// TIA Portal V20 export
DATA_BLOCK "EmNodes"   // DB3
{ DB_Accessible_From_OPC_UA := 'FALSE' }
AUTHOR : ERsystem_FA2_DH. Kim
// stored: Access Published, DBAccessibleFromOPCUA false, DBAccessibleFromWebserver false, MemoryReserve 100, Namespace Unit1
   VAR
      unitStatus { ExternalWritable := 'False'} : "LAF_typeUnitStatus";   // Status of the unit
      emFeedback { ExternalWritable := 'False'} : Array[0.._.U1_NO_OF_EMs] of "LUC_typeEmFeedback";   // Status of the individual equipment modules
      emRelations : Struct
         em00 : "Unit1.type_emRelations_em0";
         em01 : "Unit1.type_emRelations_em1";
         em02 : "Unit1.type_emRelations_em2";
         em03 : "Unit1.type_emRelations_em3";
         em04 : "Unit1.type_emRelations_em4";
         em05 : "Unit1.type_emRelations_em5";
         em06 : "Unit1.type_emRelations_em6";
         em07 : "Unit1.type_emRelations_em7";
      END_STRUCT;
      emIt { S7_SetPoint := 'True'} : Array[0..13] of "LER_OEM_Data";
      enableControlInterfaces { ExternalWritable := 'False'} : "LAF_typeEnableControlInterfaces";
      oem { ExternalAccessible := 'False'; ExternalVisible := 'False'; ExternalWritable := 'False'; S7_SetPoint := 'True'} : Array[0..10] of "LER_OEM_Data";
      FATModeSelect { ExternalWritable := 'False'} : "LER_TypeFATMode_ModeSelect";
   END_VAR
   VAR RETAIN
      FATModeInterface { ExternalWritable := 'False'} : "LER_TypeFATModeInterface";
   END_VAR
   VAR
      signalStack { ExternalWritable := 'False'} : "LUC_typeSignalStackByBool";
      clock { ExternalWritable := 'False'} : "LAF_typeGlobalClockMem";
      slmRunning { S7_SetPoint := 'True'} : Bool;
      slmPowerOff { ExternalWritable := 'False'} : Bool;
      InterfaceTestMode { ExternalWritable := 'False'} : Bool;
      CapabilityModeComplete { ExternalWritable := 'False'} : Bool;
      SamplingModeComplete { ExternalWritable := 'False'} : Bool;
      stateCommandsExecute { ExternalWritable := 'False'} : Bool;
      atLeastOneDoorUnlock { ExternalWritable := 'False'} : Bool;
      SleepModeActivationTime : Time;
      DeepSleepModeActivationTime : Time;
      SleepModeChangeReq : Bool;
      DeepSleepModeChangeReq : Bool;
      WakeupRecoveryRequired : Bool;
      sleep : Struct
         State { S7_SetPoint := 'True'} : "LER_typeSleepMode";
         command { S7_SetPoint := 'True'} : "LER_typeSleep";
      END_STRUCT;
      "========Communication========" { ExternalWritable := 'False'} : Bool;
      BA010 { ExternalWritable := 'False'} : "LER_typeCommunicationReelCut";
      BA015 { ExternalWritable := 'False'} : "LER_typeCommunicationReelCut";
      BA040 { ExternalWritable := 'False'} : "LER_typeCommunicationStack";
      BA060 { S7_SetPoint := 'True'} : "LER_typeCommunicationInspection";
      "========Safety========" { ExternalWritable := 'False'} : Bool;
      devicesSummary : "LWONIK_typeDevicesStatusSummary";
      safetyZone1OpEnable { ExternalWritable := 'False'} : "LWONIK_typeSafetyZoneManualOperation";
      safetyZone2OpEnable { ExternalWritable := 'False'} : "LWONIK_typeSafetyZoneManualOperation";
      safetyZone3OpEnable { ExternalWritable := 'False'} : "LWONIK_typeSafetyZoneManualOperation";
      doorOpenRequest : Bool;
      safetyStatusZone1 { S7_SetPoint := 'True'} : "LWONIK_typeZoneStatus";
      safetyStatusZone2 { S7_SetPoint := 'True'} : "LWONIK_typeZoneStatus";
      safetyStatusZone3 { S7_SetPoint := 'True'} : "LWONIK_typeZoneStatus";
      mainOpMode : "LWONIK_typeOperationMode";
      pHmiMode { ExternalWritable := 'False'} : "LWONIK_typePhmiMode";
      scsMode { ExternalWritable := 'False'} : "LWONIK_typeScsMode";
      rcMode1 { S7_SetPoint := 'True'} : "LWONIK_typeRollChangeMode";
      rcMode2 { S7_SetPoint := 'True'} : "LWONIK_typeRollChangeMode";
      scrapBox1 { S7_SetPoint := 'True'} : "LWONIK_typeScrapBox";
      scrapBox2 { S7_SetPoint := 'True'} : "LWONIK_typeScrapBox";
      SafetySensor { S7_SetPoint := 'True'} : "LWONIK_typeSafetySensor";
      EstopStatus { ExternalWritable := 'False'} : "LWONIK_typeFromSafetyEstopStatus";
      FdoorStatus { ExternalWritable := 'False'} : "LWONIK_typeFromSafetyDoorStatus";
      fDoorDrive : "Safety.typeFDoorFunction";
      cvCoverStatus : Struct
         cvCoverOK1 { ExternalWritable := 'False'} : Bool;
         cvCoverOK2 { ExternalWritable := 'False'} : Bool;
         cvCoverAllOK { ExternalWritable := 'False'} : Bool;
         cvCoverSystemFaults { ExternalWritable := 'False'} : Bool;
      END_STRUCT;
      AllSFDoorOpen { S7_SetPoint := 'True'} : Bool;
      AllFDoorClosed : Bool;
      OpHmiOperationEnable : Bool;
      PHmiOperationEnable : Bool;
      MobilePanelConnected : Bool;
      MobilePanelPermissions : Bool;
      BA60ExternalDoorOpen : Bool;
      SS1TimeExtension : Bool;
      EnableServoAck : Bool;
      BA10SCSModeSelect : Bool;
      BA15SCSModeSelect : Bool;
      BA40SCSModeSelect : Bool;
      BA60SCSModeSelect : Bool;
      BA60LightCurtainMutingOn : Bool;
      "=======ETC========" : Bool;
      allBrakeTest { ExternalWritable := 'False'} : "LER_typeBrakeTestUnitInterface";
      booltest { S7_SetPoint := 'True'} : Array[0..15] of Bool;
      motionInterface : Struct
         Dancer : Struct
            Enable : Bool := FALSE;
            Stop : Bool := FALSE;
            Reset : Bool := FALSE;
         END_STRUCT;
         StackMain : Struct
            Calculate { ExternalAccessible := 'False'; ExternalVisible := 'False'; ExternalWritable := 'False'} : Bool;
            SemiStep { ExternalAccessible := 'False'; ExternalVisible := 'False'; ExternalWritable := 'False'} : Bool;
            FullStep { ExternalAccessible := 'False'; ExternalVisible := 'False'; ExternalWritable := 'False'} : Bool;
            SepaClean { ExternalAccessible := 'False'; ExternalVisible := 'False'; ExternalWritable := 'False'} : Bool;
            Auto { ExternalAccessible := 'False'; ExternalVisible := 'False'; ExternalWritable := 'False'} : Bool;
            StopMotion { ExternalAccessible := 'False'; ExternalVisible := 'False'; ExternalWritable := 'False'} : Bool;
            Reset { ExternalAccessible := 'False'; ExternalVisible := 'False'; ExternalWritable := 'False'} : Bool;
         END_STRUCT;
      END_STRUCT;
      FullStepRun : Bool;
      MotionRunlockBit : Bool;
      FullStepReady : Bool;
      MotionReady : Bool;
      SpecialFunctionEnable : Bool;
   END_VAR
BEGIN
   // emRelations.em04."Bool"[10] : EM4 Motion Ready / No Job Active
   // emRelations.em04.sequence.Spare1.preOperationCheck.Bool12 : EM4 Ready For Motion
   // emRelations.em05."Bool"[10] : EM5 Motion Ready / No Job Active
   // emRelations.em05.sequence.Spare1.preOperationCheck.Bool12 : EM5 Ready For Motion
   // emRelations.em06.sequence.Spare1.preOperationCheck.Bool12 : EM6 Ready For Motion
   // emRelations.em06.sequence.Spare1.jobInterface[14].motionRequest : SepaCleanMotion Request
   // emRelations.em07."Bool"[1] : SepaGirpperAxisX Move To BA60
   // BA010.ReelCutToStack.InterfaceData."Bool"[0] : Load Enable
   // BA010.ReelCutToStack.InterfaceData."Bool"[1] : Load Complete Comfirm
   // BA010.ReelCutToStack.InterfaceData."Bool"[2] : Cell Data Report
   // BA010.ReelCutToStack.InterfaceData."Bool"[10] : CollisionAreaOn
   // BA010.ReelCutToStack.InterfaceData."Bool"[11] : CollisionAreaOff
   // BA010.ReelCutToStack.InterfaceData."Bool"[20] : Motion Ready
   // BA010.ReelCutToStack.InterfaceData."Bool"[21] : Motion Auto Standby
   // BA010.ReelCutToStack.InterfaceData."Bool"[22] : Motion Auto Mode
   // BA010.ReelCutToStack.InterfaceData."Bool"[23] : Motion Stop CMD (Motion Stop Req)
   // BA010.ReelCutToStack.InterfaceData."Bool"[30] : HoursTestMode.On/Off.Status (ReelCut)
   // BA010.ReelCutToStack.InterfaceData."Bool"[31] : HourTestMode_Completed (ReelCut)
   // BA010.ReelCutToStack.InterfaceData."Bool"[32] : CapabilityMode.On/Off.Status (ReelCut)
   // BA010.ReelCutToStack.InterfaceData."Bool"[33] : CapabilityMode_Completed (ReelCut)
   // BA010.ReelCutToStack.InterfaceData."Bool"[34] : FATMode.Apply (ReelCut)
   // BA010.ReelCutToStack.InterfaceData.LReal[10] : Select Hours (ReelCut)
   // BA010.StackToReelCut.InterfaceData."Bool"[0] : From Load Requset
   // BA010.StackToReelCut.InterfaceData."Bool"[1] : From Load Busy
   // BA010.StackToReelCut.InterfaceData."Bool"[2] : From Load Complete
   // BA010.StackToReelCut.InterfaceData."Bool"[3] : Cell Data Request
   // BA010.StackToReelCut.InterfaceData."Bool"[4] : Cell Data Report Ack
   // BA010.StackToReelCut.InterfaceData."Bool"[5] : Cell Data Report Nck
   // BA010.StackToReelCut.InterfaceData."Bool"[10] : Stack#1 Gauge RnR Complete
   // BA010.StackToReelCut.InterfaceData."Bool"[15] : HeartBeat
   // BA010.StackToReelCut.InterfaceData."Bool"[19] : From Stack#1 Count Mismatch Call
   // BA010.StackToReelCut.InterfaceData."Bool"[20] : From Motion Ready Status (Stack#1 Full)
   // BA010.StackToReelCut.InterfaceData."Bool"[21] : From Stack#1 in Motion Auto Standby
   // BA010.StackToReelCut.InterfaceData."Bool"[22] : From Stack#1 in Motion Auto Mode
   // BA010.StackToReelCut.InterfaceData."Bool"[23] : From Motion Start CMD (Stack#1 Motion Req)
   // BA010.StackToReelCut.InterfaceData."Bool"[24] : From Motion Stop CMD (Stack#1 Error)
   // BA010.StackToReelCut.InterfaceData."Bool"[25] : From Stack#1 Unloading
   // BA010.StackToReelCut.InterfaceData."Bool"[26] : From Stack#1 Loading Ok
   // BA010.StackToReelCut.InterfaceData."Bool"[30] : HoursTestMode.On/Off.Status (STK)
   // BA010.StackToReelCut.InterfaceData."Bool"[31] : HourTestMode_Completed (STK)
   // BA010.StackToReelCut.InterfaceData."Bool"[32] : CapabilityMode.On/Off.Status (STK)
   // BA010.StackToReelCut.InterfaceData."Bool"[33] : CapabilityMode_Completed (STK)
   // BA010.StackToReelCut.InterfaceData."Bool"[34] : FATMode.Apply (STK)
   // BA010.StackToReelCut.InterfaceData."Bool"[40] : HoursTestMode.On/Off.Status (INS)
   // BA010.StackToReelCut.InterfaceData."Bool"[41] : HourTestMode_Completed (INS)
   // BA010.StackToReelCut.InterfaceData."Bool"[42] : CapabilityMode.On/Off.Status (INS)
   // BA010.StackToReelCut.InterfaceData."Bool"[43] : CapabilityMode_Completed (INS)
   // BA010.StackToReelCut.InterfaceData."Bool"[44] : FATMode.Apply (INS)
   // BA010.StackToReelCut.InterfaceData.LReal[0] : From Stack#1 Cell Count
   // BA010.StackToReelCut.InterfaceData.LReal[1] : From Stack#1 CPM
   // BA010.StackToReelCut.InterfaceData.LReal[2] : Stack#1 Gauge RnR3 Mode Count
   // BA010.StackToReelCut.InterfaceData.LReal[10] : Select Hours (STK)
   // BA010.StackToReelCut.InterfaceData.LReal[11] : Select Hours (INS)
   // BA015.ReelCutToStack.InterfaceData."Bool"[0] : Load Enable
   // BA015.ReelCutToStack.InterfaceData."Bool"[1] : Load Complete Comfirm
   // BA015.ReelCutToStack.InterfaceData."Bool"[2] : Cell Data Report
   // BA015.ReelCutToStack.InterfaceData."Bool"[10] : CollisionAreaOn
   // BA015.ReelCutToStack.InterfaceData."Bool"[11] : CollisionAreaOff
   // BA015.ReelCutToStack.InterfaceData."Bool"[20] : Motion Ready
   // BA015.ReelCutToStack.InterfaceData."Bool"[21] : Motion Auto Standby
   // BA015.ReelCutToStack.InterfaceData."Bool"[22] : Motion Auto Mode
   // BA015.ReelCutToStack.InterfaceData."Bool"[23] : Motion Stop CMD (Motion Stop Req)
   // BA015.ReelCutToStack.InterfaceData."Bool"[30] : HoursTestMode.On/Off.Status (ReelCut)
   // BA015.ReelCutToStack.InterfaceData."Bool"[31] : HourTestMode_Completed (ReelCut)
   // BA015.ReelCutToStack.InterfaceData."Bool"[32] : CapabilityMode.On/Off.Status (ReelCut)
   // BA015.ReelCutToStack.InterfaceData."Bool"[33] : CapabilityMode_Completed (ReelCut)
   // BA015.ReelCutToStack.InterfaceData."Bool"[34] : FATMode.Apply (ReelCut)
   // BA015.ReelCutToStack.InterfaceData.LReal[10] : Select Hours (ReelCut)
   // BA015.StackToReelCut.InterfaceData."Bool"[0] : From Load Requset
   // BA015.StackToReelCut.InterfaceData."Bool"[1] : From Load Busy
   // BA015.StackToReelCut.InterfaceData."Bool"[2] : From Load Complete
   // BA015.StackToReelCut.InterfaceData."Bool"[3] : Cell Data Request
   // BA015.StackToReelCut.InterfaceData."Bool"[4] : Cell Data Report Ack
   // BA015.StackToReelCut.InterfaceData."Bool"[5] : Cell Data Report Nck
   // BA015.StackToReelCut.InterfaceData."Bool"[10] : Stack#1 Gauge RnR Complete
   // BA015.StackToReelCut.InterfaceData."Bool"[15] : HeartBeat
   // BA015.StackToReelCut.InterfaceData."Bool"[19] : From Stack#1 Count Mismatch Call
   // BA015.StackToReelCut.InterfaceData."Bool"[20] : From Motion Ready Status (Stack#1 Full)
   // BA015.StackToReelCut.InterfaceData."Bool"[21] : From Stack#1 in Motion Auto Standby
   // BA015.StackToReelCut.InterfaceData."Bool"[22] : From Stack#1 in Motion Auto Mode
   // BA015.StackToReelCut.InterfaceData."Bool"[23] : From Motion Start CMD (Stack#1 Motion Req)
   // BA015.StackToReelCut.InterfaceData."Bool"[24] : From Motion Stop CMD (Stack#1 Error)
   // BA015.StackToReelCut.InterfaceData."Bool"[25] : From Stack#1 Unloading
   // BA015.StackToReelCut.InterfaceData."Bool"[26] : From Stack#1 Loading Ok
   // BA015.StackToReelCut.InterfaceData."Bool"[30] : HoursTestMode.On/Off.Status (STK)
   // BA015.StackToReelCut.InterfaceData."Bool"[31] : HourTestMode_Completed (STK)
   // BA015.StackToReelCut.InterfaceData."Bool"[32] : CapabilityMode.On/Off.Status (STK)
   // BA015.StackToReelCut.InterfaceData."Bool"[33] : CapabilityMode_Completed (STK)
   // BA015.StackToReelCut.InterfaceData."Bool"[34] : FATMode.Apply (STK)
   // BA015.StackToReelCut.InterfaceData."Bool"[40] : HoursTestMode.On/Off.Status (INS)
   // BA015.StackToReelCut.InterfaceData."Bool"[41] : HourTestMode_Completed (INS)
   // BA015.StackToReelCut.InterfaceData."Bool"[42] : CapabilityMode.On/Off.Status (INS)
   // BA015.StackToReelCut.InterfaceData."Bool"[43] : CapabilityMode_Completed (INS)
   // BA015.StackToReelCut.InterfaceData."Bool"[44] : FATMode.Apply (INS)
   // BA015.StackToReelCut.InterfaceData.LReal[0] : From Stack#1 Cell Count
   // BA015.StackToReelCut.InterfaceData.LReal[1] : From Stack#1 CPM
   // BA015.StackToReelCut.InterfaceData.LReal[2] : Stack#1 Gauge RnR3 Mode Count
   // BA015.StackToReelCut.InterfaceData.LReal[10] : Select Hours (STK)
   // BA015.StackToReelCut.InterfaceData.LReal[11] : Select Hours (INS)
   // BA060.InspectionToStack.InterfaceData."Bool"[0] : Heartbeat
   // BA060.InspectionToStack.InterfaceData."Bool"[1] : ReadyForOperation
   // BA060.InspectionToStack.InterfaceData."Bool"[2] : ReachedHome
   // BA060.InspectionToStack.InterfaceData."Bool"[3] : MachineInOperation
   // BA060.InspectionToStack.InterfaceData."Bool"[4] : LoaderOutsideModule
   // BA060.InspectionToStack.InterfaceData."Bool"[5] : LoaderOutsideCollision
   // BA060.InspectionToStack.InterfaceData."Bool"[10] : PartClamped
   // BA060.InspectionToStack.InterfaceData."Bool"[11] : PartUnclamped
   // BA060.InspectionToStack.InterfaceData."Bool"[16] : RequestUnclamp
   // BA060.InspectionToStack.InterfaceData."Bool"[17] : PartOn
   // BA060.InspectionToStack.InterfaceData."Bool"[18] : RequestPart
   // BA060.InspectionToStack.InterfaceData."Bool"[19] : OnPositionUnloading
   // BA060.InspectionToStack.InterfaceData."Bool"[22] : RequestCollisionON
   // BA060.InspectionToStack.InterfaceData."Bool"[23] : UnoadComplete
   // BA060.InspectionToStack.InterfaceData."Bool"[26] : DataCatchUp
   // BA060.InspectionToStack.InterfaceData."Bool"[27] : DataCompareOK
   // BA060.InspectionToStack.InterfaceData."Bool"[28] : DataDeleted
   // BA060.InspectionToStack.InterfaceData."Bool"[32] : NG RequestPart
   // BA060.InspectionToStack.InterfaceData."Bool"[33] : NG RequestUnclamp
   // BA060.InspectionToStack.InterfaceData."Bool"[34] : NG UnoadComplete
   // BA060.InspectionToStack.InterfaceData."Bool"[40] : HoursTestMode.On/Off.Status (INS)
   // BA060.InspectionToStack.InterfaceData."Bool"[41] : HourTestMode_Completed (INS)
   // BA060.InspectionToStack.InterfaceData."Bool"[42] : CapabilityMode.On/Off.Status (INS)
   // BA060.InspectionToStack.InterfaceData."Bool"[43] : CapabilityMode_Completed (INS)
   // BA060.InspectionToStack.InterfaceData."Bool"[44] : FATMode.Apply (INS)
   // BA060.InspectionToStack.InterfaceData."Bool"[48] : ReturnToHome
   // BA060.InspectionToStack.InterfaceData."Bool"[49] : AutoStart
   // BA060.InspectionToStack.InterfaceData."Bool"[50] : EndOfCycle
   // BA060.InspectionToStack.InterfaceData."Bool"[51] : RequestGateOpen
   // BA060.InspectionToStack.InterfaceData.LReal[0] : Select Hours (INS)
   // BA060.StackToInspection.InterfaceData."Bool"[0] : Heartbeat
   // BA060.StackToInspection.InterfaceData."Bool"[1] : ReadyForOperation
   // BA060.StackToInspection.InterfaceData."Bool"[2] : ReachedHome
   // BA060.StackToInspection.InterfaceData."Bool"[3] : MachineInOperation
   // BA060.StackToInspection.InterfaceData."Bool"[4] : NoInterference
   // BA060.StackToInspection.InterfaceData."Bool"[10] : PartClamped
   // BA060.StackToInspection.InterfaceData."Bool"[11] : PartUnclamped
   // BA060.StackToInspection.InterfaceData."Bool"[16] : RequestClamp
   // BA060.StackToInspection.InterfaceData."Bool"[17] : PartOn
   // BA060.StackToInspection.InterfaceData."Bool"[18] : PartReady
   // BA060.StackToInspection.InterfaceData."Bool"[19] : LoaderInTranferArea
   // BA060.StackToInspection.InterfaceData."Bool"[20] : CollisionAreaOn
   // BA060.StackToInspection.InterfaceData."Bool"[21] : CollisionAreaOff
   // BA060.StackToInspection.InterfaceData."Bool"[23] : LoadComplete
   // BA060.StackToInspection.InterfaceData."Bool"[26] : DataCatchUp
   // BA060.StackToInspection.InterfaceData."Bool"[27] : DataCompareOK
   // BA060.StackToInspection.InterfaceData."Bool"[28] : DataDeleted
   // BA060.StackToInspection.InterfaceData."Bool"[32] : NG PartReady
   // BA060.StackToInspection.InterfaceData."Bool"[33] : NG RequestClamp
   // BA060.StackToInspection.InterfaceData."Bool"[34] : NG LoadComplete
   // BA060.StackToInspection.InterfaceData."Bool"[35] : HoursTestMode.On/Off.Status (ReelCut)
   // BA060.StackToInspection.InterfaceData."Bool"[36] : HourTestMode_Completed (ReelCut)
   // BA060.StackToInspection.InterfaceData."Bool"[37] : CapabilityMode.On/Off.Status (ReelCut)
   // BA060.StackToInspection.InterfaceData."Bool"[38] : CapabilityMode_Completed (ReelCut)
   // BA060.StackToInspection.InterfaceData."Bool"[39] : FATMode.Apply (ReelCut)
   // BA060.StackToInspection.InterfaceData."Bool"[40] : HoursTestMode.On/Off.Status (STK)
   // BA060.StackToInspection.InterfaceData."Bool"[41] : HourTestMode_Completed (STK)
   // BA060.StackToInspection.InterfaceData."Bool"[42] : CapabilityMode.On/Off.Status (STK)
   // BA060.StackToInspection.InterfaceData."Bool"[43] : CapabilityMode_Completed (STK)
   // BA060.StackToInspection.InterfaceData."Bool"[44] : FATMode.Apply (STK)
   // BA060.StackToInspection.InterfaceData."Bool"[48] : ReturnToHome
   // BA060.StackToInspection.InterfaceData."Bool"[49] : AutoStart
   // BA060.StackToInspection.InterfaceData."Bool"[50] : EndOfCycle
   // BA060.StackToInspection.InterfaceData."Bool"[51] : StopForOpenGate
   // BA060.StackToInspection.InterfaceData.LReal[0] : Select Hours (STK)
   // BA060.StackToInspection.InterfaceData.LReal[1] : Select Hours (ReelCut)
   booltest[2] := TRUE;
END_DATA_BLOCK
